PROGRAM DLOG_RRD_DEMO
VAR
	RTC_2 : RTC_2;
	CLK_PRG: CLK_PRG;
	cur_dt : DT;
	rtc_set : BOOL := TRUE;
	enable : BOOL := TRUE;
	DLOG_STORE_RRD : DLOG_STORE_RRD;
	trig_t : UDINT := 0;
	trig_m : BOOL;

	rrd_error_c : DWORD;
	rrd_error_t : BYTE;
	rrd_enable : BOOL := TRUE;
	rrd_url : T_MaxString := 'http://xxx.com/myhouse/rrd/test_rrd.php?rrd_db=test.rrd&value=';
	rrd_timeout: TIME := t#5s;

	x : DLOG_DATA;
	x1 : DLOG_DINT;
	x2 : DLOG_DINT;
	x3 : DLOG_REAL;
	x4 : DLOG_REAL;
	x5 : DLOG_REAL;
	x6 : DLOG_REAL;
	x7 : DLOG_REAL;

	GEN_SIN_1 : GEN_SIN;
	GEN_SIN_2 : GEN_SIN;
	GEN_SIN_3 : GEN_SIN;
	GEN_RMP_1: GEN_RMP;
	GEN_RMP_2: GEN_RMP;
END_VAR
VAR // added by the converter: edge detectors and wires of the graphical bodies
    _w1, _w2, _w3 : ANY;
END_VAR

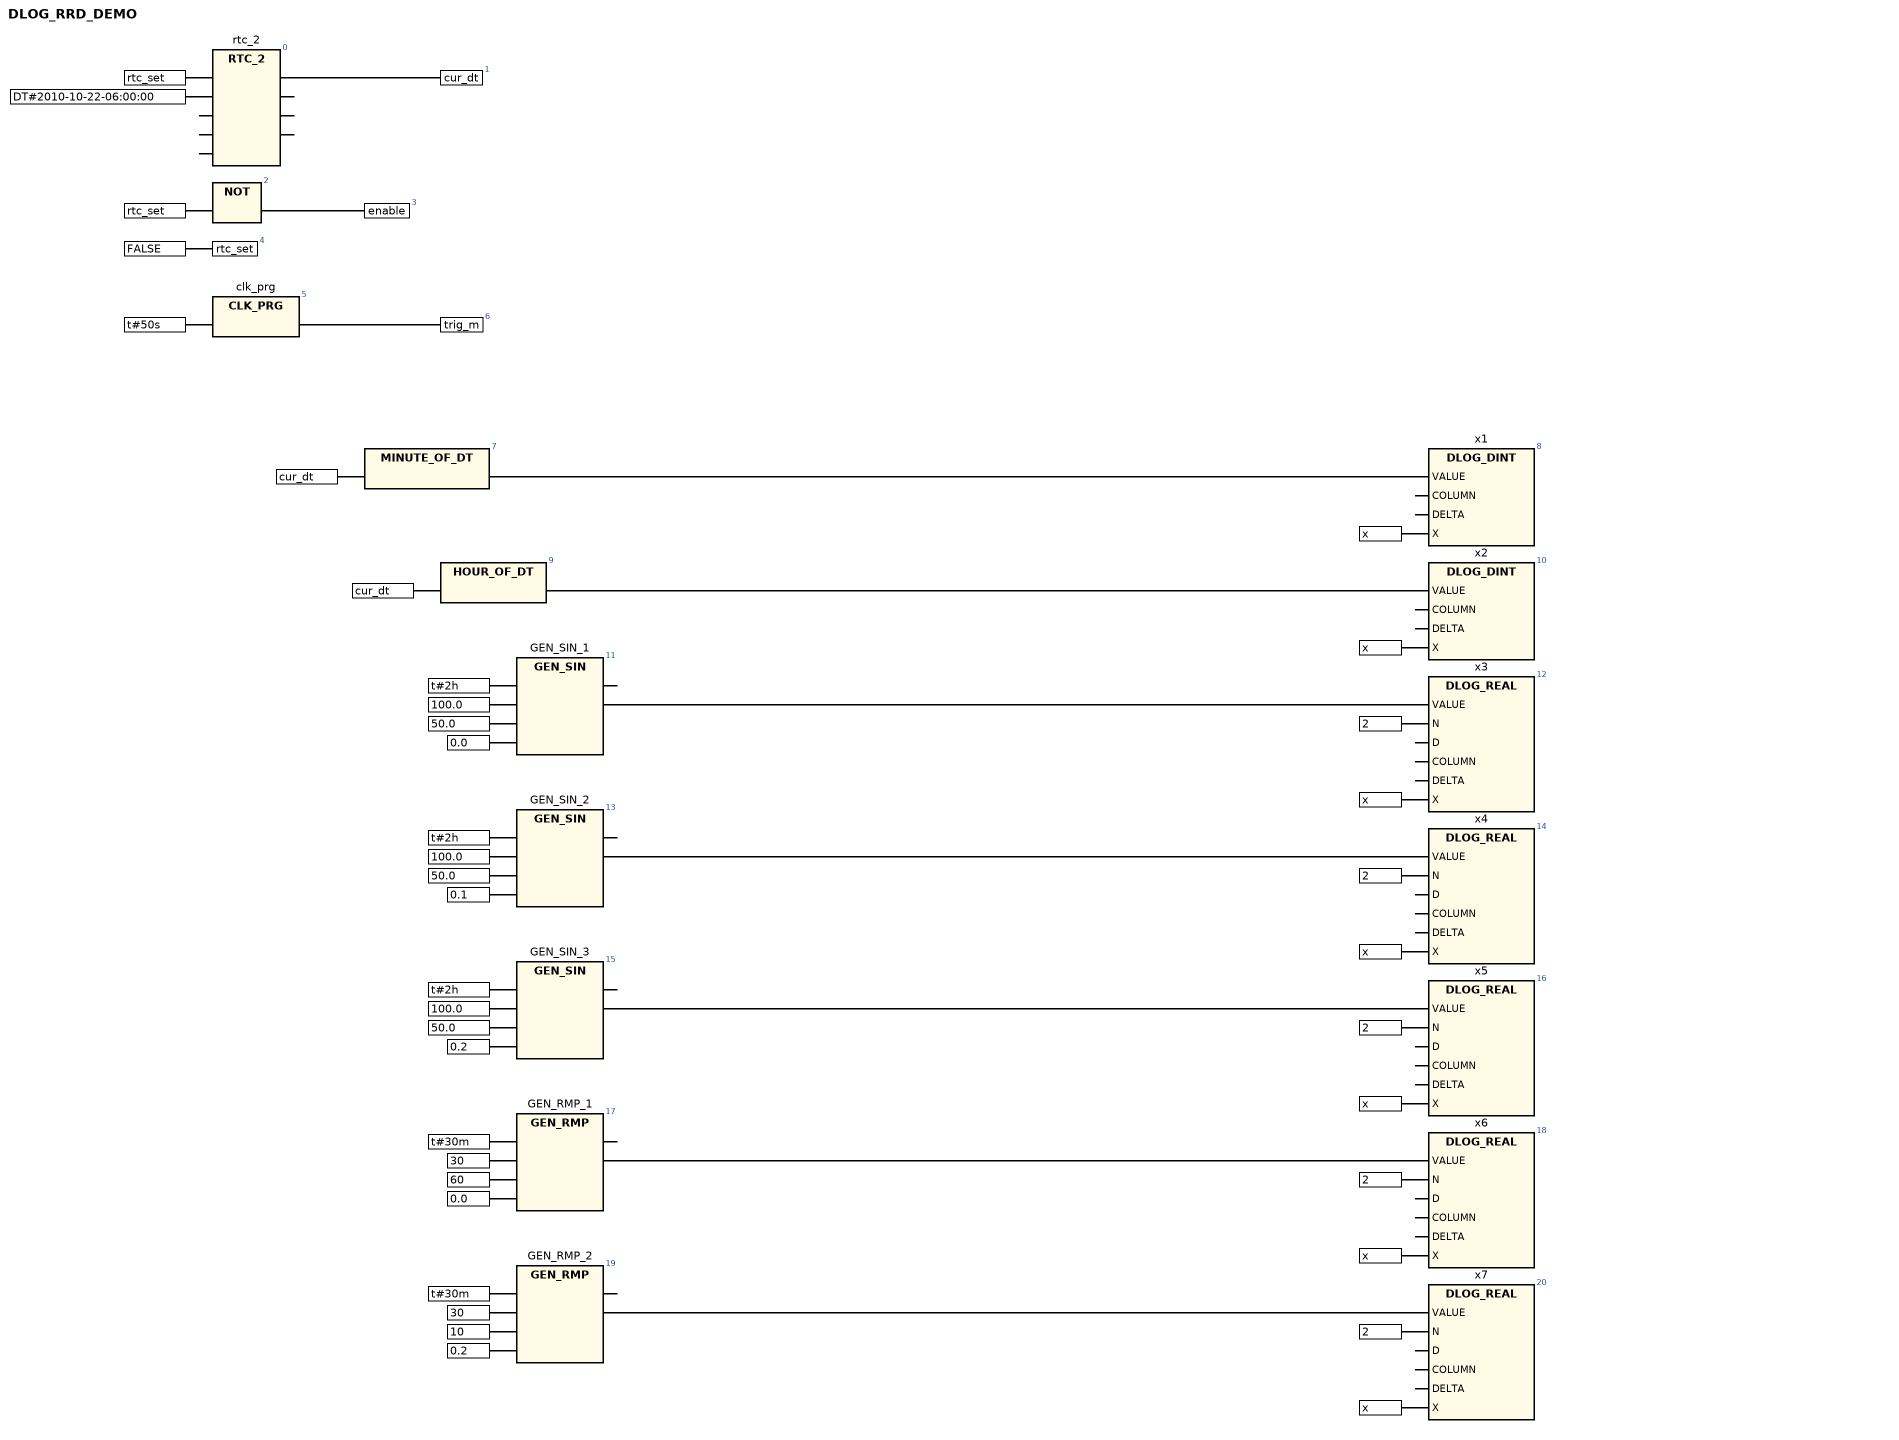
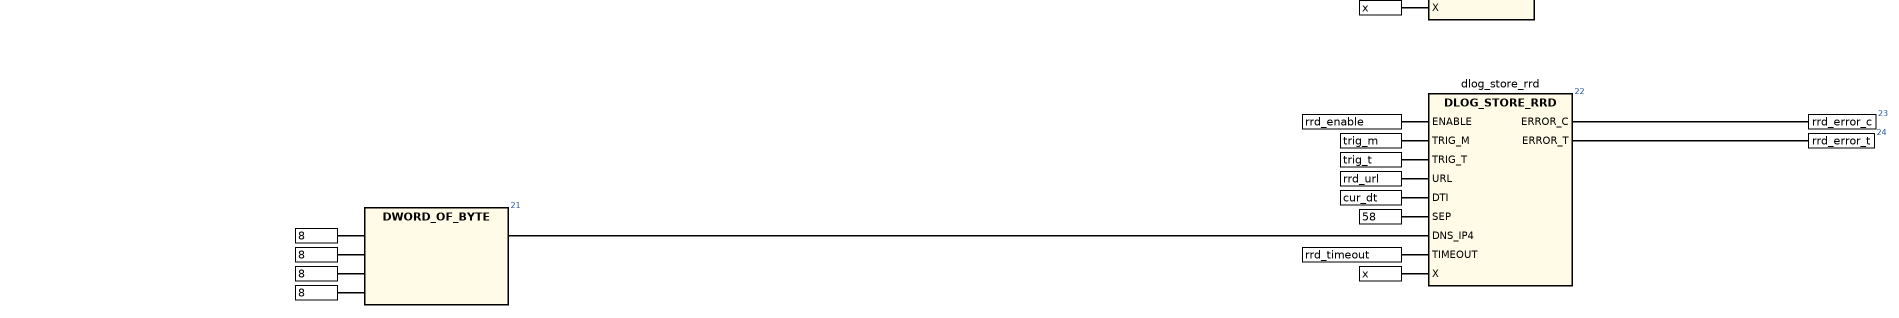
rtc_2(_in1 := rtc_set, _in2 := DT#2010-10-22-06:00:00);
cur_dt := rtc_2._out1;
enable := NOT rtc_set;
rtc_set := FALSE;
clk_prg(_in1 := t#50s);
trig_m := clk_prg._out1;
_w1 := MINUTE_OF_DT(cur_dt);
x1(VALUE := _w1, X := x); // DLOG_DINT
_w2 := HOUR_OF_DT(cur_dt);
x2(VALUE := _w2, X := x); // DLOG_DINT
GEN_SIN_1(_in1 := t#2h, _in2 := 100.0, _in3 := 50.0, _in4 := 0.0); // GEN_SIN
x3(VALUE := GEN_SIN_1._out2, N := 2, X := x); // DLOG_REAL
GEN_SIN_2(_in1 := t#2h, _in2 := 100.0, _in3 := 50.0, _in4 := 0.1); // GEN_SIN
x4(VALUE := GEN_SIN_2._out2, N := 2, X := x); // DLOG_REAL
GEN_SIN_3(_in1 := t#2h, _in2 := 100.0, _in3 := 50.0, _in4 := 0.2); // GEN_SIN
x5(VALUE := GEN_SIN_3._out2, N := 2, X := x); // DLOG_REAL
GEN_RMP_1(_in1 := t#30m, _in2 := 30, _in3 := 60, _in4 := 0.0); // GEN_RMP
x6(VALUE := GEN_RMP_1._out2, N := 2, X := x); // DLOG_REAL
GEN_RMP_2(_in1 := t#30m, _in2 := 30, _in3 := 10, _in4 := 0.2); // GEN_RMP
x7(VALUE := GEN_RMP_2._out2, N := 2, X := x); // DLOG_REAL
_w3 := DWORD_OF_BYTE(8, 8, 8, 8);
dlog_store_rrd(
    ENABLE := rrd_enable,
    TRIG_M := trig_m,
    TRIG_T := trig_t,
    URL := rrd_url,
    DTI := cur_dt,
    SEP := 58,
    DNS_IP4 := _w3,
    TIMEOUT := rrd_timeout,
    X := x);
rrd_error_c := dlog_store_rrd.ERROR_C;
rrd_error_t := dlog_store_rrd.ERROR_T;

END_PROGRAM

(* stored: Version 1.1.0.1, ProductVersion 3.1.4024.9
   POU DLOG_RRD_DEMO: Id {56a6d97f-6661-4b08-9fbe-b4f8429f1b9e}, SpecialFunc None *)
